Staubli VAL3: sendStatus.pgx

program sendStatus(string message (dimensions=1), num sio_ID (dimensions=1))
  local num asciiMessage[64]
  local num stringPos
begin
  //**************************************************
  // Method to report status of a command through: a) the TCP socket,
  // including a trailing ';' and also printing the status to the
  // screen of the MCP
  //**************************************************

  // Convert message to a ASCII code with a trailing ; to confirm the end of the message
  // The for loop is inclusive, so we go to len(message)-1 ...
  for stringPos=0 to (len(message)-1)
    asciiMessage[stringPos]=asc(message,stringPos)
  endFor
  // ... and as the string position starts at 0, we have to add the ; at the len(message) position
  asciiMessage[len(message)]=asc(";",0)

  // Print status and send message
  put("Status: ")
  putln(message)
  putln(" ")
  sioSet(sioASCII[sio_ID],asciiMessage)
end
